(* PLC project Unnamed, Unknown Unnamed 1 *)
(* stored: creationDateTime 2025-06-21T02:22:39, modificationDateTime 2025-06-21T03:07:24 *)

PROGRAM ctu_pou
  VAR
    input1 AT %IX100.0 : BOOL;
    input2 AT %IX100.1 : BOOL;
    reset AT %IX100.2 : BOOL;
    output1 AT %QX100.0 : BOOL;
    output2 AT %QX100.1 : BOOL;
  END_VAR
  VAR
    TON0 : TON;
    TOF0 : TOF;
    TP0 : TP;
    R_TRIG0 : R_TRIG;
    CTU0 : CTU;
  END_VAR
  VAR  (* added by the conversion: wires and edge detectors of the diagram *)
    R_TRIG1 : R_TRIG;
  END_VAR

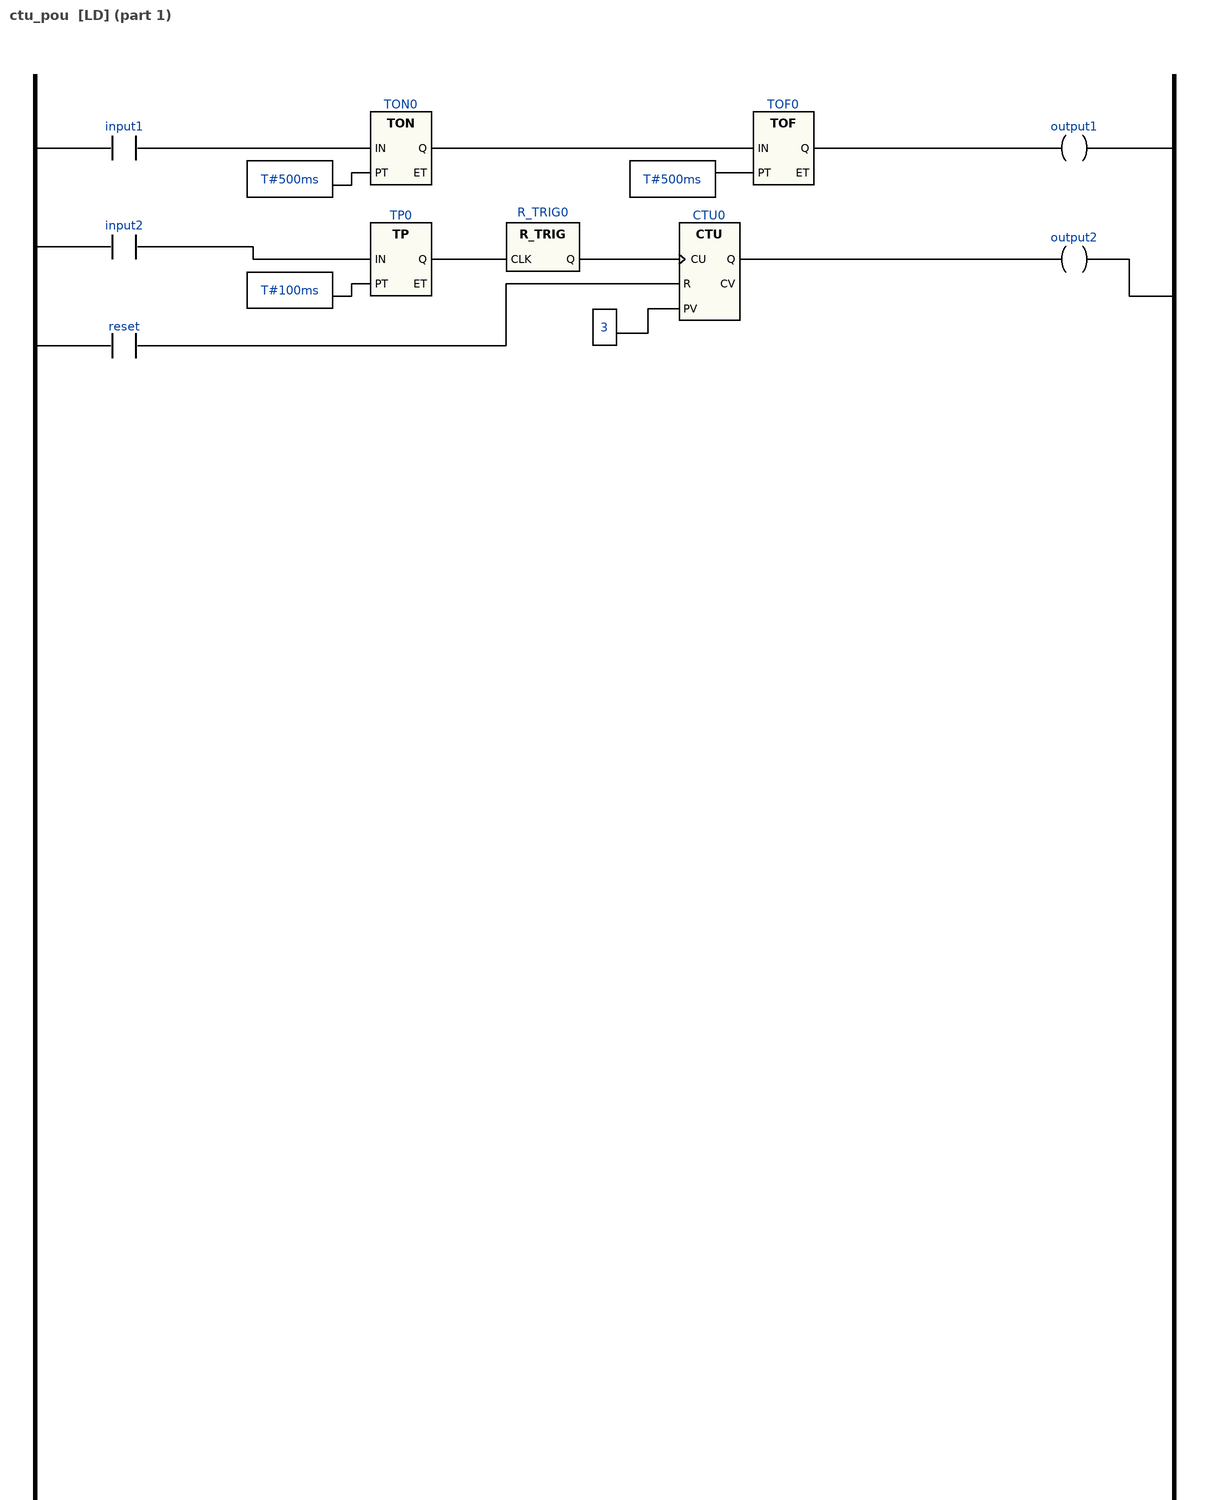
(* LD diagram, written out as Structured Text *)
TON0(IN := input1, PT := T#500ms);
TOF0(IN := TON0.Q, PT := T#500ms);
output1 := TOF0.Q;
TP0(IN := input2, PT := T#100ms);
R_TRIG0(CLK := TP0.Q);
R_TRIG1(CLK := R_TRIG0.Q);
CTU0(CU := R_TRIG1.Q, R := reset, PV := 3);
output2 := CTU0.Q;
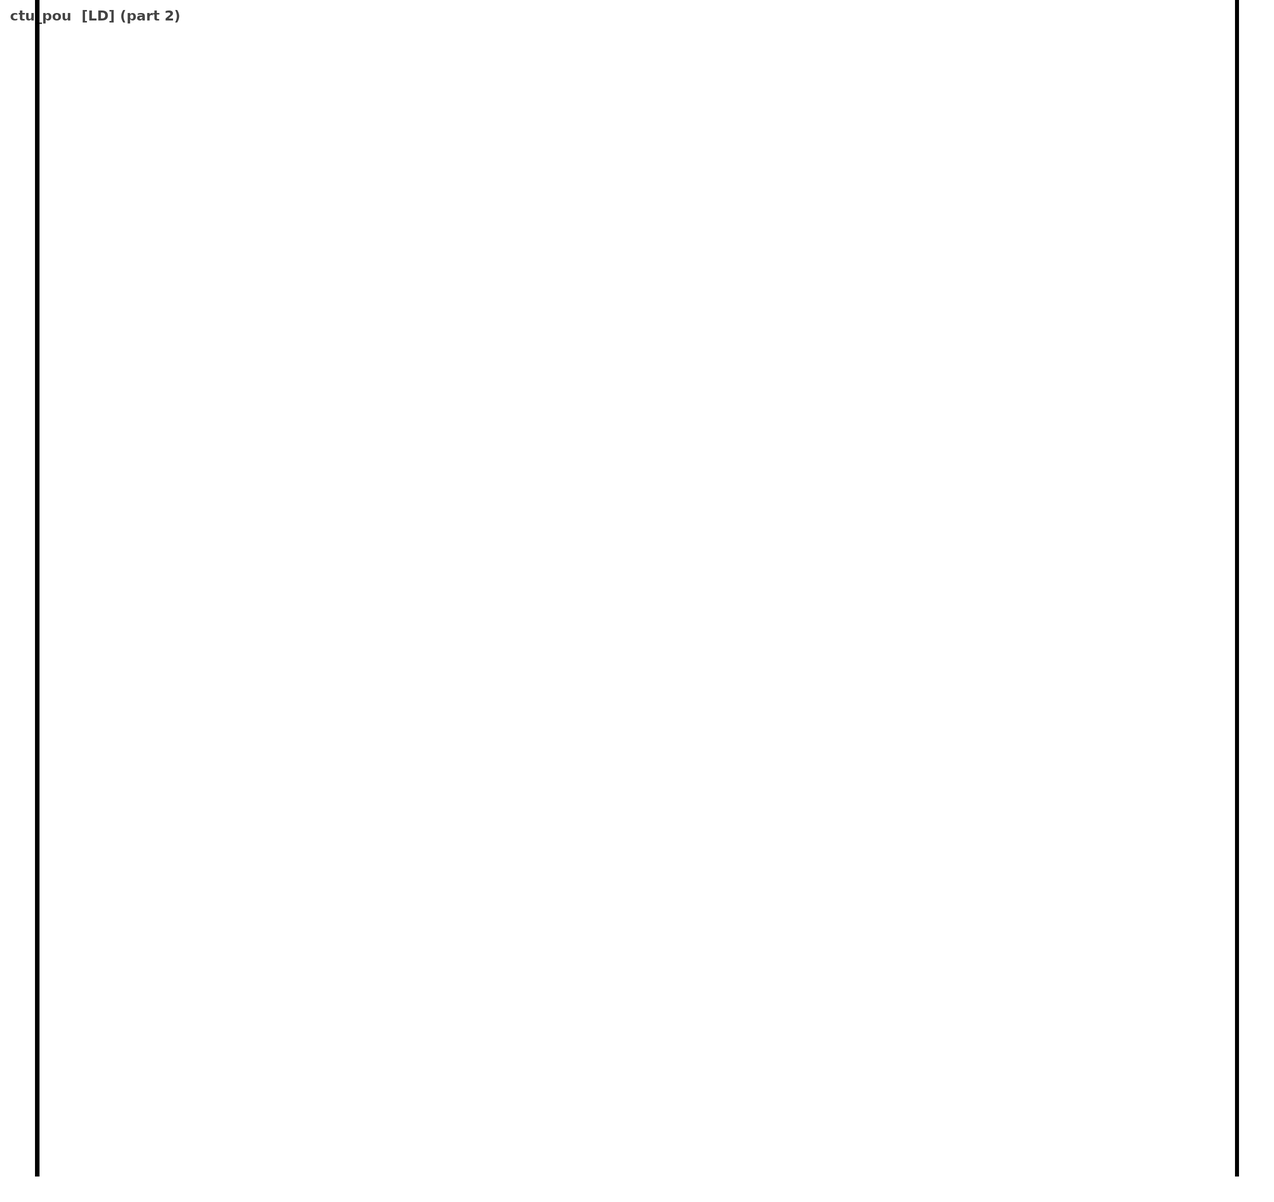
END_PROGRAM

CONFIGURATION Config0
  RESOURCE Res0 ON PLC
    TASK task0(INTERVAL := T#20ms, PRIORITY := 0);
    PROGRAM instance0 WITH task0 : ctu_pou;
  END_RESOURCE
END_CONFIGURATION
